FUNCTION_BLOCK FB_simulatedpompdigin IMPLEMENTS ITF_pompdigin
VAR
	internalState : bool;
END_VAR

{warning 'Add method implementation '}
METHOD get : BOOL
VAR_INPUT
	state	: BOOL;
END_VAR
get := internalState;
END_METHOD

END_FUNCTION_BLOCK

(* stored: Version 1.1.0.1, ProductVersion 3.1.4026.8
   POU FB_simulatedpompdigin: Id {a4b60bd1-8614-431c-a953-f3fcc946e2f0}, SpecialFunc None
   Method get: Id {30a0210a-53ae-4199-9024-345a136663b0} *)
